INTERFACE I_Nodes

METHOD PUBLIC Accept
VAR_INPUT
	Visitor : I_NodeVisitor;
END_VAR
END_METHOD

METHOD AddNode
VAR_INPUT
	Node : I_Node;
END_VAR
END_METHOD

METHOD PUBLIC TryGetNodeById : BOOL
VAR_INPUT
	Id : T_MAXSTRING;
	Destination : REFERENCE TO I_Node;
END_VAR
END_METHOD

END_INTERFACE

(* stored: Version 1.1.0.1, ProductVersion 3.1.4024.12
   Itf I_Nodes: Id {392c64f5-5891-454a-8914-1c3b0985521e}
   Method Accept: Id {307e1582-48a6-4469-a16e-3cf2e607637f}
   Method AddNode: Id {0d8acc7d-480d-4b45-9cea-d79555d4f11d}
   Method TryGetNodeById: Id {75fa4ac1-ec52-4391-8cfc-253437da3dcb} *)
